TYPE ST_MM_Header :
STRUCT
	StartBytes	:WORD :=16#ABBA;
	MsgLength	:BYTE :=0;
END_STRUCT
END_TYPE

(* stored: Version 1.1.0.1, ProductVersion 3.1.4020.12
   DUT ST_MM_Header: Id {35c87d0b-424e-4d78-9d2d-224bdd667129} *)
